PROGRAM MAIN
VAR
END_VAR

TcUnit.RUN();

END_PROGRAM

(* stored: Version 1.1.0.1, ProductVersion 3.1.4024.6
   POU MAIN: Id {7558137b-b54e-4a00-bef4-79d805178012}, SpecialFunc None *)
